(*			
	RAFALOS
	Rafał Osajda		19.09.2025		TC 4024.66
	
*)
FUNCTION_BLOCK FB_BaseDescriptor IMPLEMENTS ITF_BaseDescriptor
VAR
	stDescriptor					: ST_BaseDescriptor;
END_VAR

METHOD PUBLIC GetDefaultValue : REAL
VAR_INPUT
END_VAR
GetDefaultValue			:= THIS^.stDescriptor.rDefaultValue;
END_METHOD

METHOD PUBLIC GetDefaultValueFrom : REAL
VAR_INPUT
	stIN				: ST_BaseDescriptor;
END_VAR
GetDefaultValueFrom			:= stIN.rDefaultValue;
END_METHOD

METHOD PUBLIC GetDescriptor : ST_BaseDescriptor
VAR_INPUT
END_VAR
GetDescriptor		:= this^.stDescriptor;
END_METHOD

METHOD PUBLIC GetMax : REAL
VAR_INPUT
END_VAR
GetMax					:= THIS^.stDescriptor.rMax;
END_METHOD

METHOD PUBLIC GetMaxFrom : REAL
VAR_INPUT
	stIN				: ST_BaseDescriptor;
END_VAR
GetMaxFrom				:= stIN.rMax;
END_METHOD

METHOD PUBLIC GetMin : REAL
VAR_INPUT
END_VAR
GetMin				:= THIS^.stDescriptor.rMin;
END_METHOD

METHOD PUBLIC GetMinFrom : REAL
VAR_INPUT
	stIN			: ST_BaseDescriptor;
END_VAR
GetMinFrom			:= stIN.rMin;
END_METHOD

METHOD PUBLIC GetTexts : ST_BaseLabel
VAR_INPUT
END_VAR
GetTexts				:=THIS^.stDescriptor.stTexts;
END_METHOD

METHOD PUBLIC GetTextsFrom : ST_BaseLabel
VAR_INPUT
	stIN				: ST_BaseDescriptor;
END_VAR
GetTextsFrom			:=stIN.stTexts;
END_METHOD

METHOD PUBLIC GetUnit : STRING(6)
VAR_INPUT
END_VAR
GetUnit			:= THIS^.stDescriptor.sUnit;
END_METHOD

METHOD PUBLIC GetUnitFrom : STRING(6)
VAR_INPUT
	stIN			: ST_BaseDescriptor;
END_VAR
GetUnitFrom			:= stIN.sUnit;
END_METHOD

METHOD PUBLIC GetValue : REAL
VAR_INPUT
END_VAR
GetValue			:= this^.stDescriptor.rValue;
END_METHOD

METHOD PUBLIC GetValueFrom : REAL
VAR_INPUT
	stIN			: ST_BaseDescriptor;
END_VAR
GetValueFrom		:= stIN.rValue;
END_METHOD

METHOD PUBLIC SetDefaultValue
VAR_INPUT
	rDefaultValue: REAL;
END_VAR
THIS^.stDescriptor.rDefaultValue		:= rDefaultValue;
END_METHOD

METHOD PUBLIC SetDefaultValueIn
VAR_INPUT
	stIN			: REFERENCE TO ST_BaseDescriptor;
	rDefaultValue	: REAL;
END_VAR
stIN.rDefaultValue		:= rDefaultValue;
END_METHOD

METHOD PUBLIC SetMax
VAR_INPUT
	rMax: REAL;
END_VAR
THIS^.stDescriptor.rMax		:= rMax;
END_METHOD

METHOD PUBLIC SetMaxIn
VAR_INPUT
	stIN			: REFERENCE TO ST_BaseDescriptor;
	rMax: REAL;
END_VAR
stIN.rMax		:= rMax;
END_METHOD

METHOD PUBLIC SetMin
VAR_INPUT
	rMin: REAL;
END_VAR
THIS^.stDescriptor.rMin		:= rMin;
END_METHOD

METHOD PUBLIC SetMinIn
VAR_INPUT
	stIN			: REFERENCE TO ST_BaseDescriptor;
	rMin: REAL;
END_VAR
stIn.rMin		:= rMin;
END_METHOD

METHOD PUBLIC SetText
VAR_INPUT
	eLocation			: E_BaseLocation;
	wsDescription		: WSTRING;
END_VAR
THIS^.stDescriptor.stTexts.arrText [eLocation]	:= wsDescription;
END_METHOD

METHOD PUBLIC SetTextIn
VAR_INPUT
	stIN				: REFERENCE TO ST_BaseDescriptor;
	eLocation			: E_BaseLocation;
	wsDescription		: WSTRING;
END_VAR
stIN.stTexts.arrText [eLocation]	:= wsDescription;
END_METHOD

METHOD PUBLIC SetTexts
VAR_INPUT
	stTexts				: ST_BaseLabel;
END_VAR
THIS^.stDescriptor.stTexts			:= stTexts;
END_METHOD

METHOD PUBLIC SetTextsIn
VAR_INPUT
	stIN				: REFERENCE TO ST_BaseDescriptor;
	stTexts				: ST_BaseLabel;
END_VAR
stIN.stTexts			:= stTexts;
END_METHOD

METHOD PUBLIC SetUnit
VAR_INPUT
	sUnit: STRING(6);
END_VAR
THIS^.stDescriptor.sUnit		:= sUnit;
END_METHOD

METHOD PUBLIC SetUnitIn
VAR_INPUT
	stIN			: REFERENCE TO ST_BaseDescriptor;
	sUnit: STRING(6);
END_VAR
stIN.sUnit		:= sUnit;
END_METHOD

METHOD PUBLIC SetValue
VAR_INPUT
	rValue: REAL;
END_VAR
THIS^.stDescriptor.rValue		:= rValue;
END_METHOD

METHOD PUBLIC SetValueIn
VAR_INPUT
	stIN			: REFERENCE TO ST_BaseDescriptor;
	rValue			: REAL;
END_VAR
stIN.rValue			:= rValue;
END_METHOD

END_FUNCTION_BLOCK

(* stored: Version 1.1.0.1
   POU FB_BaseDescriptor: Id {91493404-5653-0352-2d94-26778011a0ca}, SpecialFunc None
   Method GetDefaultValue: Id {7672acfb-69d1-0152-0da7-f699bf266bad}
   Method GetDefaultValueFrom: Id {93ecbc15-beae-07f7-0fee-7d8703a092f1}
   Method GetDescriptor: Id {655083d0-f571-0cef-3358-6590c9822db9}
   Method GetMax: Id {8c76e190-abee-0b2f-27c2-dfbab096def1}
   Method GetMaxFrom: Id {a5506df0-4038-0da5-194a-e313bfde06d7}
   Method GetMin: Id {1bb9af4c-532c-0d65-0fa1-3f85303ee695}
   Method GetMinFrom: Id {f119c5bf-5215-04b0-3e90-a03de3b261d5}
   Method GetTexts: Id {417909bc-3071-05d7-1b3f-8468c5f7f250}
   Method GetTextsFrom: Id {4acf1e5f-432e-00fe-0c6f-8c2f45e7aa09}
   Method GetUnit: Id {c59d07ba-453e-0fd3-241b-d8705866834f}
   Method GetUnitFrom: Id {f5c9a08d-ebc0-0203-32b8-f0e9cf2245cf}
   Method GetValue: Id {1fbad2d2-c73a-00b7-272a-3bd1a663b3de}
   Method GetValueFrom: Id {5c626a0d-81f1-07da-12a6-85eff4b1e6ea}
   Method SetDefaultValue: Id {09cf2edb-c6b5-0603-37d0-2e6642dcc45f}
   Method SetDefaultValueIn: Id {3ee9ec08-c105-0f08-284f-f5553e811f9d}
   Method SetMax: Id {0f50b22f-5dec-0af4-1e0b-94d421cf37c6}
   Method SetMaxIn: Id {e53c210a-480d-0ff4-3927-08a86a268ae7}
   Method SetMin: Id {cdcb8462-e776-0a08-04c6-034dd95fa910}
   Method SetMinIn: Id {8f149a5f-c077-01d6-158f-c2ff67bb05de}
   Method SetText: Id {3c16ad50-9b2e-080a-1ab9-d69019c1102c}
   Method SetTextIn: Id {cf04b86a-0e02-018b-326c-60ebfa4a50c3}
   Method SetTexts: Id {31ae5e96-267f-0a74-148a-8b7537ed702e}
   Method SetTextsIn: Id {78dd0fb2-206e-0adc-0dab-082cea18059a}
   Method SetUnit: Id {c7b5bc13-b76d-0bbe-0ade-846421544371}
   Method SetUnitIn: Id {867b33d2-482b-0025-30a9-c6885b6af5ec}
   Method SetValue: Id {fe9b8b66-0a69-0021-26b6-4b3d78392ea8}
   Method SetValueIn: Id {929f6494-9bbe-072d-352f-3d44ac9b3a16} *)
